TYPE DoChannel :
STRUCT
	{attribute addProperty Name "Output"}
	Output AT %Q* : BOOL;
END_STRUCT
END_TYPE

(* stored: Version 1.1.0.1, ProductVersion 3.1.4024.9
   DUT DoChannel: Id {28d65377-b1e1-0836-13ed-9f11d3939bd9} *)
